% RSLogix 500 project Compare.RSS, saved by version 8.30.00.16 %
PROJECT "UNTITLED"    % processor: Bul.1763 MicroLogix 1100 Series B %

PROGRAM FILES
  LAD 2   3 rungs

DATA FILES
  O0 OUTPUT  4 elements
  I1 INPUT  6 elements
  S2 STATUS  66 elements
  B3 BINARY  1 elements
  T4 TIMER  1 elements
  C5 COUNTER  1 elements
  R6 CONTROL  1 elements
  N7 INTEGER  1 elements
  F8 FLOAT  1 elements

LADDER 2
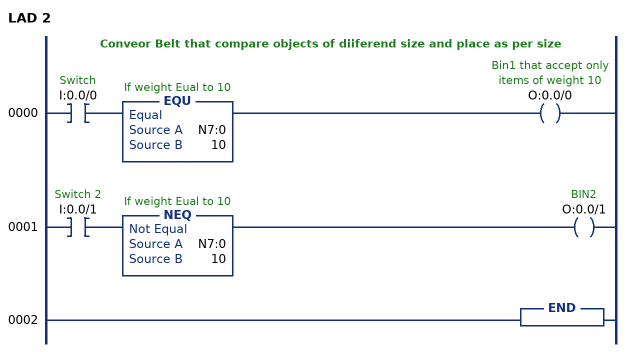
% Rung: 0 %
% TITLE: Conveor Belt that compare objects of diiferend size and place as per size %
SOR XIC I:0.0/0 EQU N7:0 10 OTE O:0.0/0 EOR
%   I:0.0/0  "Switch" %
%   N7:0  "If weight Eual to 10" %
%   O:0.0/0  "Bin1 that accept only items of weight 10" %
% Rung: 1 %
SOR XIC I:0.0/1 NEQ N7:0 10 OTE O:0.0/1 EOR
%   I:0.0/1  "Switch 2" %
%   N7:0  "If weight Eual to 10" %
%   O:0.0/1  BIN2 %
% Rung: 2 %
SOR END EOR

DATA TABLE (non-zero values as saved)
DATA N7
% N7:0 % 20
